FUNCTION_BLOCK E_RTimeOut (* Simple implementation of the timeout services *)
  (* Standard: 61499-2; Description: Copyright (c) 2017 fortiss GmbH This program and the accompanying materials are made available under the terms of the Eclipse Public License 2.0 which is available at https://www.eclipse.org/legal/epl-2.0/ SPDX-License-Identifier: EPL-2.0 *)
  (* Version 1.0, 2017-09-22, Alois Zoitl, fortiss GmbH, initial API and implementation and/or initial documentation *)
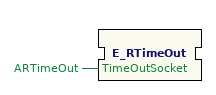
  SOCKETS
    TimeOutSocket : ARTimeOut;
  END_SOCKETS
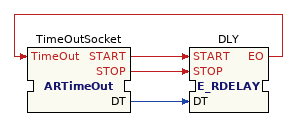
  FBS
    DLY : E_RDELAY;
  END_FBS
  EVENT_CONNECTIONS
    TimeOutSocket.START TO DLY.START;
    TimeOutSocket.STOP TO DLY.STOP;
    DLY.EO TO TimeOutSocket.TimeOut;
  END_CONNECTIONS
  DATA_CONNECTIONS
    TimeOutSocket.DT TO DLY.DT;
  END_CONNECTIONS
END_FUNCTION_BLOCK
